INTERFACE ITF_Regelschuif_OutOpen_DG

METHOD set : BOOL
VAR_INPUT
	state : BOOL;
END_VAR
END_METHOD

END_INTERFACE

(* stored: Version 1.1.0.1, ProductVersion 3.1.4026.8
   Itf ITF_Regelschuif_OutOpen_DG: Id {947359a5-030b-423b-ba13-85037873d4e2}
   Method set: Id {211449b0-b7a5-4e42-9ead-8d9108ce7609} *)
